Universal Robots PolyScope program: rotate45cw.urp

Program rotate45cw (installation=default directory=/programs createdIn=5.14.5 lastSavedIn=5.14.5 robotSerialNumber=20236801216)
Calibrated DH parameters: a=[-0.000021, -0.748897, -0.28186, -0.00004, -0.000055, 0]; d=[0.236225, -424.082933, -1564.66872, 1988.95162, 0.159094, 0.153873]; alpha=[1.570844, 0.001002, 0.000337, 1.571488, -1.569996, 0]; deltaTheta=[0, -0.516316, 5.626292, 1.173211, 0.000001, 0]
InitVariablesNode
Robot Program (runOnlyOnce=true)
  Call align_tcp_left
  Script file /programs/speedl_test.script
    | #rot_speed=0.1
    | #current_pose=get_actual_tcp_pose()
    | #time_int = 5
    | #target_pose=pose_trans(current_pose, p[0,0,0,0,0,rot_speed*time_int])
    | #speedl(pose_sub(target_pose, current_pose), rot_speed, time_int)
    | 
    | speedl([0,0,0,0,0,0.5],0.1,5)
SubProgram -> align_tcp_left
SubProgram align_tcp_left (keepSynchronizedWithDisk=false) programFile=/programs/align_tcp_left.urp
  'this program aligns the tcp parallel to the y direction'
  cp := get_actual_tcp_pose()
  aligned_y_pose := p[cp[0],cp[1],cp[2],1.570796,0,0]
  MoveJ speed 60 deg/s, acceleration 80 deg/s^2 (useActiveTCP=true) feature=Base
    Waypoint Variable (Variable): variable=aligned_y_pose
